# EPICS substitutions: apps/iocBoot/iocclassc1test/joerger_classc1.substitutions
#
# joerger_classc1.substitutions
#
# Author: Wesley Moore (wmoore@jlab.org)
# Date:   Oct 2015
#
file "$(TOP)/db/joerger.db" {
pattern {P,      S,      OUT,        DTYP,               FREQ}
        {scaler, _c,     "#C0 S0 @", "Joerger VSC8/16",  10000000}
        {scaler, _d,     "#C2 S0 @", "Joerger VSC8/16",  10000000}
        {scaler, _e,     "#C1 S0 @", "Joerger VSC8/16",  10000000}
}
